ABB RobotStudio station: Test.rsstn

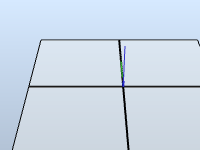
Station Station (saved by RobotStudio 6.8.8148.134)
Layout (positions relative to the parent item):
